// TwinCAT 3 PLC project TcpIp_Lib
// ProgramVersion: 3.1.4022.0
// libraries:
//   Tc2_Standard, * (Beckhoff Automation GmbH)
//   Tc2_System, * (Beckhoff Automation GmbH)
//   Tc2_TcpIp, * (Beckhoff Automation GmbH)
//   Tc3_Module, * (Beckhoff Automation GmbH)
// project tree:
//   Base Component/stream_lib/Class/Binary/ C_BINARYREADER.TcPOU, C_BINARYWRITER.TcPOU
//   Base Component/stream_lib/Class/Stream/ C_BINARYSTREAM.TcPOU
//   Base Component/stream_lib/Datatype/ E_STREAMSEEKTYPE.TcDUT
//   Base Component/stream_lib/Interface/ I_STREAM.TcIO
//   Base Component/tcp_ip/ cTcpIpClient.TcPOU
// (motion and I/O tree: see PLC project motion_library)
// real-time tasks:
//   TASK PlcTask: cycle T#10ms, priority 20, ADS port 350

// ---- Base Component/stream_lib/Datatype/E_STREAMSEEKTYPE.TcDUT
{attribute 'qualified_only'}
{attribute 'strict'}
TYPE E_STREAMSEEKTYPE :
(
	Origin := 0,
	Current,
	Current_Reversed,
	End
);
END_TYPE

// ---- Base Component/stream_lib/Interface/I_STREAM.TcIO
INTERFACE I_STREAM

PROPERTY BufferSize : UDINT
GET
END_GET
END_PROPERTY

METHOD Close : DINT
VAR_INPUT
END_VAR
END_METHOD

PROPERTY EndOfStream : BOOL
GET
END_GET
END_PROPERTY

PROPERTY IsValid : BOOL
GET
END_GET
END_PROPERTY

METHOD Peek : DINT
VAR_INPUT
	ptr_DataOut : POINTER TO BYTE;
END_VAR
END_METHOD

PROPERTY Position : UDINT
GET
END_GET
END_PROPERTY

METHOD Read : DINT
VAR_INPUT
	ptr_DataOut : PVOID;
	Length		: UDINT;
END_VAR
END_METHOD

METHOD Seek : DINT
VAR_INPUT
	Offset 		: UDINT;
	SeekStyle 	: E_STREAMSEEKTYPE;
END_VAR
END_METHOD

METHOD Write : DINT
VAR_INPUT
	ptr_DataIn	: PVOID;
	Length		: UDINT;
END_VAR
END_METHOD

END_INTERFACE

// ---- Base Component/stream_lib/Class/Binary/C_BINARYREADER.TcPOU
FUNCTION_BLOCK C_BINARYREADER
VAR_INPUT
END_VAR
VAR_OUTPUT
END_VAR
VAR
	_BASESTREAM 	: I_STREAM;
END_VAR

PROPERTY BASE_STREAM : I_STREAM
GET
Base_Stream := _BASESTREAM;
END_GET
END_PROPERTY

METHOD CLOSE : DINT
VAR_INPUT
END_VAR
Close := _BASESTREAM.Close();
_BASESTREAM := 0;
RETURN;
END_METHOD

METHOD NEW : DINT
VAR_INPUT
	STREAM : I_STREAM;
END_VAR
IF STREAM = 0 THEN
	New := 1;
	RETURN;
ELSE
	IF STREAM.IsValid THEN
		_BASESTREAM := STREAM;
		_BASESTREAM.Seek( 0, E_STREAMSEEKTYPE.Origin);
		New := -1;
		RETURN;
	ELSE
		New := 1;
		RETURN;
	END_IF
END_IF
END_METHOD

METHOD READ_BOOL : DINT
VAR_INPUT
	out_data : POINTER TO BOOL;
END_VAR
IF _BASESTREAM = 0 THEN
	Read_Bool := 1;
	RETURN;
END_IF

Read_Bool := _BASESTREAM.Read(out_data , 1);
RETURN;
END_METHOD

METHOD READ_BYTES : DINT
VAR_INPUT
	out_data 	: POINTER TO BYTE;
	length		: UDINT;
END_VAR
IF _BASESTREAM = 0 THEN
	Read_Bytes := 1;
	RETURN;
END_IF

Read_Bytes := _BASESTREAM.Read(out_data, length);
RETURN;
END_METHOD

METHOD READ_DOUBLE : DINT
VAR_INPUT
	out_data : POINTER TO LREAL;
END_VAR
IF _BASESTREAM = 0 THEN
	Read_Double := 1;
	RETURN;
END_IF

Read_Double := _BASESTREAM.Read(out_data , 8);
RETURN;
END_METHOD

METHOD READ_FLOAT : DINT
VAR_INPUT
	out_data : POINTER TO REAL;
END_VAR
IF _BASESTREAM = 0 THEN
	Read_Float := 1;
	RETURN;
END_IF

Read_Float := _BASESTREAM.Read(out_data , 4);
RETURN;
END_METHOD

METHOD READ_INT16 : DINT
VAR_INPUT
	out_data : POINTER TO INT;
END_VAR
IF _BASESTREAM = 0 THEN
	Read_Int16 := 1;
	RETURN;
END_IF

Read_Int16 := _BASESTREAM.Read(out_data , 2);
RETURN;
END_METHOD

METHOD READ_INT32 : DINT
VAR_INPUT
	out_data : POINTER TO DINT;
END_VAR
IF _BASESTREAM = 0 THEN
	Read_Int32 := 1;
	RETURN;
END_IF

Read_Int32 := _BASESTREAM.Read(out_data , 4);
RETURN;
END_METHOD

METHOD READ_STRING : DINT
VAR_INPUT
	out_data 	: PVOID;
	length		: UDINT;
END_VAR
IF _BASESTREAM = 0 THEN
	Read_String := 1;
	RETURN;
END_IF

Read_String := _BASESTREAM.Read(out_data, length);
RETURN;
END_METHOD

METHOD READ_UINT16 : DINT
VAR_INPUT
	out_data : POINTER TO UINT;
END_VAR
IF _BASESTREAM = 0 THEN
	Read_UInt16 := 1;
	RETURN;
END_IF

Read_UInt16 := _BASESTREAM.Read(out_data , 4);
RETURN;
END_METHOD

METHOD READ_UINT32 : DINT
VAR_INPUT
	out_data : POINTER TO UDINT;
END_VAR
IF _BASESTREAM = 0 THEN
	Read_UInt32 := 1;
	RETURN;
END_IF

Read_UInt32 := _BASESTREAM.Read(out_data , 4);
RETURN;
END_METHOD

END_FUNCTION_BLOCK

// ---- Base Component/stream_lib/Class/Binary/C_BINARYWRITER.TcPOU
FUNCTION_BLOCK C_BINARYWRITER
VAR_INPUT
END_VAR
VAR_OUTPUT
END_VAR
VAR
	_BASESTREAM 	: I_STREAM;
END_VAR

PROPERTY BASE_STREAM : I_STREAM
GET
Base_Stream := _BASESTREAM;
END_GET
END_PROPERTY

METHOD CLOSE : DINT
VAR_INPUT
END_VAR
Close := _BASESTREAM.Close();
_BASESTREAM := 0;
RETURN;
END_METHOD

METHOD NEW : DINT
VAR_INPUT
	STREAM : I_STREAM;
END_VAR
IF STREAM = 0 THEN
	New := 1;
	RETURN;
ELSE
	IF STREAM.IsValid THEN
		_BASESTREAM := STREAM;
		_BASESTREAM.Seek( 0, E_STREAMSEEKTYPE.Origin);
		New := -1;
		RETURN;
	ELSE
		New := 1;
		RETURN;
	END_IF
END_IF
END_METHOD

METHOD WRITE_BOOL : DINT
VAR_INPUT
	in_data : BOOL;
END_VAR
IF _BASESTREAM = 0 THEN
	Write_Bool := 1;
	RETURN;
END_IF

Write_Bool := _BASESTREAM.Write(ADR(in_data), 1);
RETURN;
END_METHOD

METHOD WRITE_BYTES : DINT
VAR_INPUT
	in_data 	: POINTER TO BYTE;
	length		: UDINT;
END_VAR
IF _BASESTREAM = 0 THEN
	Write_Bytes := 1;
	RETURN;
END_IF

Write_Bytes := _BASESTREAM.Write(in_data, length);
RETURN;
END_METHOD

METHOD WRITE_DOUBLE : DINT
VAR_INPUT
	in_data : LREAL;
END_VAR
IF _BASESTREAM = 0 THEN
	Write_Double := 1;
	RETURN;
END_IF

Write_Double := _BASESTREAM.Write(ADR(in_data), 8);
RETURN;
END_METHOD

METHOD WRITE_FLOAT : DINT
VAR_INPUT
	in_data : REAL;
END_VAR
IF _BASESTREAM = 0 THEN
	Write_Float := 1;
	RETURN;
END_IF

Write_Float := _BASESTREAM.Write(ADR(in_data) , 4);
RETURN;
END_METHOD

METHOD WRITE_INT16 : DINT
VAR_INPUT
	in_data : INT;
END_VAR
IF _BASESTREAM = 0 THEN
	Write_Int16 := 1;
	RETURN;
END_IF

Write_Int16 := _BASESTREAM.Write(ADR(in_data) , 2);
RETURN;
END_METHOD

METHOD WRITE_INT32 : DINT
VAR_INPUT
	in_data : DINT;
END_VAR
IF _BASESTREAM = 0 THEN
	Write_Int32 := 1;
	RETURN;
END_IF

Write_Int32 := _BASESTREAM.Write(ADR(in_data) , 4);
RETURN;
END_METHOD

METHOD WRITE_STRING : DINT
VAR_INPUT
	in_data 	: PVOID;
	length		: UDINT;
END_VAR
IF _BASESTREAM = 0 THEN
	Write_String := 1;
	RETURN;
END_IF

Write_String := _BASESTREAM.Write(in_data, length);
RETURN;
END_METHOD

METHOD WRITE_UINT16 : DINT
VAR_INPUT
	in_data : UINT;
END_VAR
IF _BASESTREAM = 0 THEN
	Write_UInt16 := 1;
	RETURN;
END_IF

Write_UInt16 := _BASESTREAM.Write(ADR(in_data) , 4);
RETURN;
END_METHOD

METHOD WRITE_UINT32 : DINT
VAR_INPUT
	in_data : UDINT;
END_VAR
IF _BASESTREAM = 0 THEN
	Write_UInt32 := 1;
	RETURN;
END_IF

Write_UInt32 := _BASESTREAM.Write(ADR(in_data) , 4);
RETURN;
END_METHOD

END_FUNCTION_BLOCK

// ---- Base Component/stream_lib/Class/Stream/C_BINARYSTREAM.TcPOU
FUNCTION_BLOCK C_BINARYSTREAM IMPLEMENTS I_STREAM
VAR_INPUT
END_VAR
VAR_OUTPUT
END_VAR
VAR
	_MEMBUFFER 	: POINTER TO BYTE;
	_POSITION	: UDINT;
	//_PERMISSIBLE_LIMIT 		: UDINT;
	_MEMSIZE	: UDINT;
END_VAR

PROPERTY BUFFER_SIZE : UDINT
GET
Buffer_Size := _MEMSIZE;
END_GET
END_PROPERTY

METHOD CLOSE : DINT
VAR_INPUT
END_VAR
IF _MEMBUFFER <> 0 THEN
	__DELETE(_MEMBUFFER);
	_MEMBUFFER := 0;
END_IF
_POSITION := 0;
_PERMISSIBLE_LIMIT := 0;
_MEMSIZE := 0;
END_METHOD

PROPERTY END_OF_STREAM : BOOL
GET
IF _MEMBUFFER <> 0 THEN
	End_Of_Stream := _POSITION >= _MEMSIZE;
ELSE
	End_Of_Stream := TRUE;
END_IF
END_GET
END_PROPERTY

METHOD FB_exit : BOOL
VAR_INPUT
	bInCopyCode : BOOL; // if TRUE, the exit method is called for exiting an instance that is copied afterwards (online change).
END_VAR
IF NOT bInCopyCode THEN
    CLOSE();
END_IF
END_METHOD

PROPERTY IS_VALID : BOOL
GET
Is_Valid := _MEMBUFFER <> 0;
END_GET
END_PROPERTY

METHOD NEW : DINT
VAR_INPUT
	StreamSize	: UDINT;
END_VAR
IF _MEMBUFFER <> 0 THEN
	__DELETE(_MEMBUFFER);
END_IF
_MEMSIZE 				:= StreamSize;
//_PERMISSIBLE_LIMIT	 	:= _MEMSIZE - 1;
_POSITION 				:= 0;
_MEMBUFFER 				:= __NEW(BYTE, _MEMSIZE);

New := -1;
RETURN;
END_METHOD

METHOD PEEK : DINT
VAR_INPUT
	ptr_DataOut	: POINTER TO BYTE;
END_VAR
IF EndOfStream THEN
	Peek := 1; 
	RETURN;
ELSE
	ptr_DataOut^ := _MEMBUFFER[_POSITION];
	Peek := -1;
	RETURN;
END_IF
END_METHOD

PROPERTY POSITION : UDINT
GET
POSITION := _POSITION;
END_GET
END_PROPERTY

METHOD READ : DINT
VAR_INPUT
	ptr_DataOut	: PVOID;
	Length		: UDINT;
END_VAR
IF End_Of_Stream THEN
	Read := 1;
	RETURN;
ELSE
	IF _POSITION + Length > _MEMSIZE THEN
		Read := 2;
		RETURN;
	ELSE
		MEMCPY(ptr_DataOut, _MEMBUFFER + _POSITION, Length);
		_POSITION := _POSITION + Length;
		Read := -1;
		RETURN;
	END_IF
END_IF
END_METHOD

METHOD SEEK : DINT
VAR_INPUT
	Offset		: UDINT;	//Permissible range is 0 upto the total buffer size - 1;
	SeekStyle	: E_STREAMSEEKTYPE;
END_VAR
CASE SeekStyle OF 
	//Offsets from the beginning of the stream
	E_STREAMSEEKTYPE.Origin:
		IF Offset > _MEMSIZE THEN
			Seek := 1;
			RETURN;
		ELSE
			_POSITION := Offset;
			Seek := -1;
			RETURN;
		END_IF
	//Offsets from the end of the stream
	E_STREAMSEEKTYPE.End:
		IF Offset > _MEMSIZE THEN
			Seek := 1;
			RETURN;
		ELSE
			_POSITION := (_MEMSIZE) - Offset;
			Seek := -1;
			RETURN;
		END_IF
	//Offsets from the current position of the stream
	E_STREAMSEEKTYPE.Current:
		IF _POSITION + Offset > _MEMSIZE THEN
			Seek := 1;
			RETURN;
		ELSE
			_POSITION := _POSITION + Offset;
			Seek := -1;
			RETURN;
		END_IF
	//Offsets from the current position of the stream
	E_STREAMSEEKTYPE.Current_Reversed:
		IF Offset > _POSITION  THEN
			Seek := 1;
			RETURN;
		ELSE
			_POSITION := _POSITION - Offset;
			Seek := -1;
			RETURN;
		END_IF
END_CASE
END_METHOD

METHOD WRITE : DINT
VAR_INPUT
	ptr_DataIn	: PVOID;
	Length		: UDINT;
END_VAR
IF End_Of_Stream THEN
	Write := 1;
	RETURN;
ELSE
	IF _POSITION + Length > _MEMSIZE THEN
		Write := 2;
		RETURN;
	ELSE
		MEMCPY(_MEMBUFFER + _POSITION, ptr_DataIn, Length);
		_POSITION := _POSITION + Length;
		Write := -1;
		RETURN;
	END_IF
END_IF
END_METHOD

END_FUNCTION_BLOCK

// ---- Base Component/tcp_ip/cTcpIpClient.TcPOU
FUNCTION_BLOCK cTcpIpClient
VAR_INPUT
END_VAR
VAR_OUTPUT
END_VAR
VAR
	fbSocketOpen 	: FB_SocketConnect;
	fbSocketClose	: FB_SocketClose;
	fbSnd			: FB_SocketSend;
	fbRcv			: FB_SocketReceive;
	
	_socket_		: T_HSOCKET;
	_timeout_		: TIME := T#3S;
	_bufferSize_	: UDINT := 4096;
	_clientbuffer 	: C_BINARYSTREAM;
	
	_fragment_		: ARRAY[0..511] OF BYTE;
	_rcv_poll_		: Ton := (PT := T#100MS);
END_VAR
VAR CONSTANT
	_RETURN_CODE_ERROR_ 		: DINT := 1;
	_RETURN_CODE_ERROR_NO_DATA_ : DINT := 100;
	_RETURN_CODE_ERROR_OVERRANGE_ : DINT := 101;
	_RETURN_CODE_BUSY_ : DINT := 0;
	_RETURN_CODE_SUCCESS_ : DINT := -1;
END_VAR

IF (_socket_.handle <> 0) THEN
	_rcv_poll_(IN:=TRUE);
	fbRcv(
		sSrvNetId:= , 
		hSocket:= _socket_, 
		cbLen:= 512, 
		pDest:= ADR(_fragment_), 
		bExecute:= TRUE, 
		tTimeout:= _timeout_, 
		bBusy=> , 
		bError=> , 
		nErrId=> , 
		nRecBytes=> );
	IF fbRcv.bError THEN
		fbRcv(bExecute := FALSE);
		_rcv_poll_(IN:=FALSE);
	ELSIF NOT fbRcv.nRecBytes <> 0 THEN
		fbRcv(bExecute := FALSE);
		_rcv_poll_(IN:=FALSE);
		_clientbuffer.WRITE(ADR(_fragment_), fbRcv.nRecBytes);
	ELSIF _rcv_poll_.Q THEN
		_rcv_poll_(IN:=FALSE);
	END_IF
ELSE
	_rcv_poll_(IN:=FALSE);
END_IF

PROPERTY available : bool
GET
available := _clientbuffer.Position <> 0;
END_GET
END_PROPERTY

METHOD connect : dint
VAR_INPUT
	host : STRING(15);
	port : UDINT;
END_VAR
fbSocketOpen(
	sSrvNetId:= , 
	sRemoteHost:= host, 
	nRemotePort:= port, 
	bExecute:= TRUE, 
	tTimeout:= _timeout_, 
	bBusy=> , 
	bError=> , 
	nErrId=> , 
	hSocket=> );
IF fbSocketOpen.bError THEN
	fbSocketOpen (bExecute := FALSE);
	connect := _RETURN_CODE_ERROR_;
	RETURN;
ELSIF NOT fbSocketOpen.bBusy THEN
	_socket_ := fbSocketOpen.hSocket;
	fbSocketOpen (bExecute := FALSE);
	connect := _RETURN_CODE_SUCCESS_;
	RETURN;
ELSE
	connect := _RETURN_CODE_BUSY_;
	RETURN;
END_IF
END_METHOD

METHOD destroy : dint
VAR_INPUT
END_VAR
fbSocketClose(
	sSrvNetId:= , 
	hSocket:= _socket_, 
	bExecute:= TRUE, 
	tTimeout:= , 
	bBusy=> , 
	bError=> , 
	nErrId=> );
IF fbSocketClose.bError THEN
	fbSocketClose( bExecute:= FALSE );
	destroy := _RETURN_CODE_ERROR_;
	RETURN;
ELSIF NOT fbSocketClose.bBusy THEN
	memset(ADR(_socket_), 0, SIZEOF(_socket_));
	fbSocketClose( bExecute:= FALSE );
	destroy := _RETURN_CODE_SUCCESS_;
	RETURN;
END_IF
destroy := _RETURN_CODE_BUSY_;
RETURN;
END_METHOD

METHOD FB_exit : BOOL
VAR_INPUT
	bInCopyCode : BOOL; // if TRUE, the exit method is called for exiting an instance that is copied afterwards (online change).
END_VAR
_clientbuffer.CLOSE();
END_METHOD

METHOD FB_init : BOOL
VAR_INPUT
	bInitRetains : BOOL; // if TRUE, the retain variables are initialized (warm start / cold start)
	bInCopyCode : BOOL;  // if TRUE, the instance afterwards gets moved into the copy code (online change)
END_VAR
_clientbuffer.NEW(_bufferSize_);
END_METHOD

METHOD read : dint
VAR_INPUT
	pOut 	: PVOID;
	length	: UDINT;
END_VAR
IF NOT available THEN
	read := _RETURN_CODE_ERROR_NO_DATA_;
ELSE
	IF _clientbuffer.SEEK(length, E_STREAMSEEKTYPE.Current_Reversed) > 0 THEN
		read := _RETURN_CODE_ERROR_OVERRANGE_;
		RETURN;
	ELSE
		CASE _clientbuffer.READ(pOut, length) OF 
			1,2:
				read := _RETURN_CODE_ERROR_OVERRANGE_;
				RETURN;
			-1:
				_clientbuffer.SEEK(length, E_STREAMSEEKTYPE.Current_Reversed);
				read := _RETURN_CODE_SUCCESS_;
				RETURN;
		END_CASE
	END_IF
END_IF
END_METHOD

METHOD send : DINT
VAR_INPUT
	pData : PVOID;
	length: udint;
END_VAR
IF pData = 0 OR length = 0 THEN
	send := _RETURN_CODE_ERROR_;
	RETURN;
END_IF

fbSnd(
	sSrvNetId:= , 
	hSocket:= _socket_, 
	cbLen:= length, 
	pSrc:= pData, 
	bExecute:= TRUE, 
	tTimeout:= _timeout_, 
	bBusy=> , 
	bError=> , 
	nErrId=> );
IF fbSnd.bError THEN
	fbSnd(bExecute := FALSE);
	send := _RETURN_CODE_ERROR_;
	RETURN;
ELSIF NOT fbSnd.bBusy THEN 
	fbSnd(bExecute := FALSE);
	send := _RETURN_CODE_SUCCESS_;
	RETURN;
END_IF
send := _RETURN_CODE_BUSY_;
RETURN;
END_METHOD

END_FUNCTION_BLOCK
